PROGRAM DehumidifierControl
VAR_INPUT
	// enable signal for der Dehumidifier
	Enable:	BOOL := TRUE;
	// manual enable signal
	ManualEnable: BOOL;
END_VAR
VAR
	// run dehumidifer at last for n seconds to avoid fast switching cycles
	HumidityTrigger: SR;
	RunDelay : TON := (PT:=T#30S);
	ManualTimer: TON := (PT := T#3H);
	LowOverride: TON := (PT := T#3H);
	// classic event log
	DehumidifierLog: FB_EventLog;
	
	OnTrigger:	R_TRIG;
	OffTrigger:	F_TRIG;
END_VAR
VAR CONSTANT
	HumidityBayLow:		REAL := 65.0;
	HumidityBayHigh:	REAL := 75.0;
END_VAR

HumidityTrigger( SET1 := ManualEnable OR 
						LowOverride.Q OR
						(Enable AND Environment.HumidityBay > HumidityBayHigh),
				RESET := Environment.HumidityBay < HumidityBayLow);
// override if we stay above low limit for too long
LowOverride( In := Environment.HumidityBay > HumidityBayLow);
				
// deactivate Manual Signal aftern n hours
ManualTimer( IN := ManualEnable);
IF ManualTimer.Q AND ManualEnable THEN
	ManualEnable := FALSE;
END_IF

// delay switch on to avoid overload
RunDelay(IN := HumidityTrigger.Q1);
GVL_Environment.Dehumidifier := RunDelay.Q;

DehumidifierLog(Trigger := GVL_Environment.Dehumidifier, OnMessage := 'The dehumidifier is on.', OffMessage := 'The dehumidifier is off.');

(*** MQTT Section ***)
OnTrigger(CLK := GVL_Environment.Dehumidifier);
OffTrigger(CLK := GVL_Environment.Dehumidifier);
IF OnTrigger.Q OR OffTrigger.Q THEN
	MAIN.MQTTClient.Publish('bay', 'bay', 'Dehumidifier', BOOL_TO_STRING(GVL_Environment.Dehumidifier));
END_IF

END_PROGRAM

(* stored: Version 1.1.0.1, ProductVersion 3.1.4024.9
   POU DehumidifierControl: Id {a196ab05-b1bb-47c7-be4b-4d1ebd710b0e}, SpecialFunc None *)
